{attribute 'Tc2GvlVarNames'}
VAR_CONFIG
END_VAR

(* stored: Version 1.1.0.1, ProductVersion 3.1.4022.10
   GVL Variablen_Konfiguration: Id {784502fa-227e-4dfb-ac7d-63a01a768db2} *)
